FUNCTION_BLOCK STRUCT_DEMUX (* Service Interface Function Block Type *)
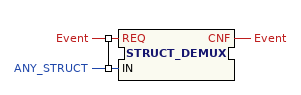
  EVENT_INPUT
    REQ WITH IN; (* Normal Execution Request *)
  END_EVENT
  EVENT_OUTPUT
    CNF; (* Execution Confirmation *)
  END_EVENT
  VAR_INPUT
    IN : ANY_STRUCT;
  END_VAR
END_FUNCTION_BLOCK
